PROGRAM MAIN
VAR
	idxState AT%I* :WORD;
	idxInput AT%I*	:BYTE;
	idxModeDisplay AT%I*:BYTE;
	idxerror AT%I*	:WORD;
	idxerrorSent :WORD :=0;
	idxControl AT%I*	:WORD;
	
	fbMessage : FB_TcMessage;
	EnableEventSent : BOOL :=TRUE;
	MovementFinishedEventSent :BOOL := FALSE;
	
	
	Linear: AXIS_REF;
	count :INT;
	fbAxisPower: MC_Power;
    fbAxisMoveAbsolute: MC_MoveAbsolute;
	fbAxisMoveRel: MC_MoveRelative;
	fbMcHome: MC_Home;
	fbReset: MC_Reset;
    bEnable: BOOL := FALSE;
    fOverride: LREAL := 100;
    bMove: BOOL := FALSE;
    fTargetPosition: LREAL := 90;
    fTargetVelocity: LREAL := 50;
	home :BOOL:=FALSE;
	resetAxis :BOOL:=FALSE;
	TestingMode: BOOL := FALSE;


	(* fbMqttClient : FB_IotMqttClient;
	SetParameter : BOOL :=TRUE;
	mqttConnect : BOOL :=TRUE;
	(*publish settings*)
	TopicPub   : STRING(255) := 'PLC';
    PayloadPub : STRING(255);
	MQTTi :UDINT;
	

	 (* received message *)
    Subscribed    : BOOL;
    TopicSub      : STRING(255) := 'PLC/Telemetry';
    {attribute 'TcEncoding':='UTF-8'}
    sTopicRcv      : STRING(255);
    {attribute 'TcEncoding':='UTF-8'}
    sPayloadRcv    : STRING(255);
    fbMessageQueue : FB_IotMqttMessageQueue;
    fbMessage      : FB_IotMqttMessage;
	
	fbMQTTtimer : TON :=(PT:=T#1S);
	*)
	
	

	
	

	TestPosA: REAL :=200;
	TestPosB: REAL :=100;
	MoveAbsDone: BOOL := TRUE;
	TestingFlag: BOOL := FALSE;
	TestingActive:BOOL :=FALSE;
	Estop: BOOL;
	TestingTime: TON:=(pt:=T#5S);
	ResetConfirmation: BOOL;
END_VAR

Linear.ReadStatus();

Estop :=  NOT idxinput.3;

IF Estop THEN  //Estop check
	bEnable:=FALSE;
END_IF

IF NOT (idxerror = idxerrorSent) THEN
	idxerrorSent:= idxerror;
	fbMessage.CreateEx(TC_Events.LinearMotor.IDXmotorError,0);
	fbMessage.ipArguments.Clear().AddDWord(idxerror);
	fbMessage.Send(0);
END_IF

// Events Handling enable Motor 
IF bEnable = EnableEventSent THEN	
	EnableEventSent := NOT EnableEventSent;
IF bEnable THEN
	fbMessage.CreateEx(TC_Events.LinearMotor.Motor_enabled,0);
ELSE
	fbMessage.CreateEx(TC_Events.LinearMotor.Motor_disabled,0);
END_IF
fbMessage.Send(0);
END_IF



fbAxisPower(
    Axis:= Linear,
    Enable:= bEnable,
    Enable_Positive:= bEnable,
    Enable_Negative:= bEnable,
    Override:= fOverride
  );

// move Absolute Axis

	fbAxisMoveAbsolute(
    Axis:= Linear,
    Execute:= bMove,
    Position:= fTargetPosition,
    Velocity:= fTargetVelocity);
	IF bMove THEN
	fbMessage.CreateEx(TC_Events.LinearMotor.MotorMove,0);
	fbMessage.ipArguments.Clear();
	fbMessage.ipArguments.AddLReal(fTargetPosition);
	fbMessage.ipArguments.AddLReal(fTargetVelocity);
	fbMessage.Send(0);
	MovementFinishedEventSent:= FALSE;
	bMove := FALSE;

ELSIF fbAxisMoveAbsolute.Done AND NOT MovementFinishedEventSent THEN
	fbMessage.CreateEx(TC_Events.LinearMotor.MoveComplete,0);
	fbMessage.Send(0);
	MovementFinishedEventSent := TRUE;
	
END_IF



	
// Home Axis
	fbMcHome(
	Axis:=Linear,
	Execute:=home,
	Position:=510,
	HomingMode:=MC_DefaultHoming);
IF home THEN
	fbMessage.CreateEx(TC_Events.LinearMotor.Homing,0);
	fbMessage.Send(0);
	home:= FALSE;	
END_IF

	

	
IF resetAxis THEN
fbReset(
Axis:=Linear,
Execute:=TRUE,
Done =>ResetConfirmation);
resetAxis:=FALSE;
idxControl := 16#80;// restop linear Motor
fbMessage.CreateEx(TC_Events.LinearMotor.AxisReset,0);
fbMessage.send(0);
END_IF

	
IF TestingMode AND Linear.NcToPlc.StateDword.0 THEN //in testing mode
	IF linear.NcToPlc.AxisState=0 AND NOT fbAxisMoveAbsolute.Busy THEN// check if axis has no current jobs 
		bMove:=TRUE;
	END_IF
	
	IF  fbAxisMoveAbsolute.Done THEN//swap ends for test
		TestingFlag := NOT TestingFlag;
	END_IF

	IF TestingFlag THEN// change targets 
		fTargetPosition:= TestPosA;
	ELSE 
		fTargetPosition:= TestPosB;
	END_IF
	
END_IF

END_PROGRAM

(* stored: Version 1.1.0.1, ProductVersion 3.1.4024.11
   POU MAIN: Id {4e8483c1-ccbb-4128-b543-7a53eb2e77a5}, SpecialFunc None *)
